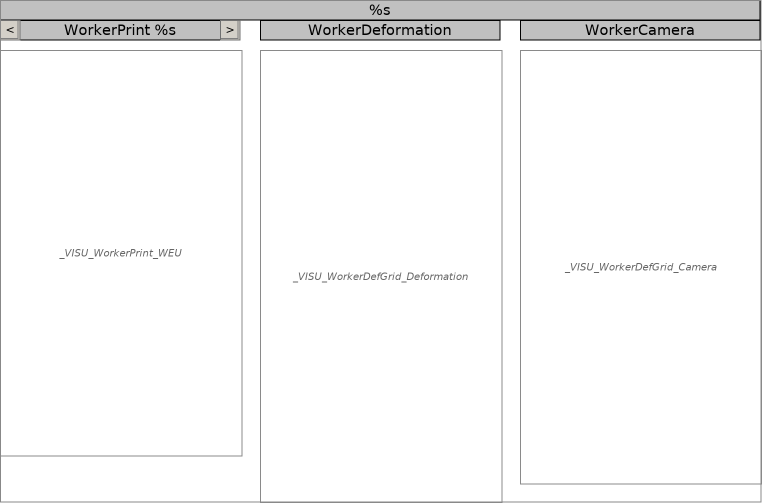
VISUALIZATION _VISU_Pm_Worker  // 762x503
VAR_IN_OUT
	mInst : FB_PrintModule_WEU;
END_VAR
    Frame (0,50 242x406)
        shows _VISU_WorkerPrint_WEU(m_Inst := mInst.fbWorkerPrint[1])
    Rectangle (0,20 240x20), "WorkerPrint %s", text variable: mInst.fbView.nSelWorkerPrint
    Frame (520,50 242x434)
        shows _VISU_WorkerDefGrid_Camera(m_Inst := mInst.fbWorkerCamera)
    Rectangle (520,20 240x20), "WorkerCamera"
    Rectangle (0,0 760x20), "%s", text variable: mInst.fbAdsPm.aO_Name
    Rectangle (260,20 240x20), "WorkerDeformation"
    Frame (260,50 242x453)
        shows _VISU_WorkerDefGrid_Deformation(m_Inst := mInst.fbWorkerDeformation)
    Button (0,20 20x20), "<"
        OnMouseClick: execute { mInst.fbView.nSelWorkerPrint := mInst.fbView.nSelWorkerPrint - 1; }
    Button (220,20 20x20), ">"
        OnMouseClick: execute { mInst.fbView.nSelWorkerPrint := mInst.fbView.nSelWorkerPrint + 1; }
END_VISUALIZATION

(* stored: Version 1.1.0.1, ProductVersion 3.1.4024.11
   Visu _VISU_Pm_Worker: Id {978ceb48-7732-4238-8bf1-4a3c5db6e0e2} *)
